FUNCTION FUN_Compare_Timestructs : SINT //returns: 1 IF ts1 is older, -1 if ts2 is older, 0 if equal
VAR_INPUT
	ts1	:	TIMESTRUCT;
	ts2	:	TIMESTRUCT;
END_VAR
VAR
END_VAR

//OUTPUT: 1 IF ts1 is older, -1 if ts2 is older, 0 if equal
IF (ts1.wYear=ts2.wYear) THEN
	IF (ts1.wMonth=ts2.wMonth) THEN
		IF (ts1.wDay=ts2.wDay) THEN
			IF (ts1.wHour=ts2.wHour) THEN
				IF (ts1.wMinute=ts2.wMinute) THEN
					IF (ts1.wSecond=ts2.wSecond) THEN
						IF (ts1.wMilliseconds=ts2.wMilliseconds) THEN
							FUN_Compare_Timestructs:=0;
						ELSIF (ts1.wMilliseconds>ts2.wMilliseconds) THEN
								FUN_Compare_Timestructs:=-1;
						ELSE
								FUN_Compare_Timestructs:=1;
						END_IF
						
					ELSIF (ts1.wSecond>ts2.wSecond) THEN
						FUN_Compare_Timestructs:=-1;
					ELSE
						FUN_Compare_Timestructs:=1;
					END_IF
					
				ELSIF (ts1.wMinute>ts2.wMinute) THEN
					FUN_Compare_Timestructs:=-1;
				ELSE
					FUN_Compare_Timestructs:=1;
				END_IF
				
			ELSIF (ts1.wHour>ts2.wHour) THEN
				FUN_Compare_Timestructs:=-1;
			ELSE
				FUN_Compare_Timestructs:=1;
			END_IF
		
		ELSIF (ts1.wDay>ts2.wDay) THEN
			FUN_Compare_Timestructs:=-1;
		ELSE
			FUN_Compare_Timestructs:=1;
		END_IF
	
	ELSIF (ts1.wMonth>ts2.wMonth) THEN
		FUN_Compare_Timestructs:=-1;
	ELSE
		FUN_Compare_Timestructs:=1;
	END_IF
	
ELSIF (ts1.wYear>ts2.wYear) THEN
	FUN_Compare_Timestructs:=-1;
ELSE
	FUN_Compare_Timestructs:=1;
END_IF

END_FUNCTION

(* stored: Version 1.1.0.1, ProductVersion 3.1.4024.12
   POU FUN_Compare_Timestructs: Id {8ceaed40-c670-442d-a26c-7437ae3662f6}, SpecialFunc None *)
